FUNCTION_BLOCK FB_AddMcsAxesXyzToMcGroup
VAR_IN_OUT
	stAxis				: ARRAY[1..3] OF AXIS_REF;	
	stGroupRef			: AXES_GROUP_REF;
END_VAR
VAR_INPUT
	bExecute				: BOOL;
END_VAR
VAR_OUTPUT
	bDone				: BOOL;
	bBusy				: BOOL;
	bError				: BOOL;
END_VAR
VAR
	fbAddAxis			: ARRAY[1..3] OF MC_AddAxisToGroup;
	i					: UINT;
END_VAR

bDone := TRUE;
bBusy := FALSE;
bError := FALSE;

fbAddAxis[1].IdentInGroup := MCS_X; //X-Axis
fbAddAxis[2].IdentInGroup := MCS_Y; //Y-Axis
fbAddAxis[3].IdentInGroup := MCS_Z; //Z-Axis

FOR i:=1 TO 3 DO
	fbAddAxis[i](AxesGroup:=stGroupRef, Axis := stAxis[i], Execute := bExecute);

	IF (NOT fbAddAxis[i].Done) THEN
		bDone := FALSE;
	END_IF
	IF (fbAddAxis[i].Busy) THEN
		bBusy := TRUE;
	END_IF
	IF (fbAddAxis[i].Error) THEN
		bError := TRUE;
	END_IF
END_FOR

END_FUNCTION_BLOCK

(* stored: Version 1.1.0.1, ProductVersion 3.1.4024.5
   POU FB_AddMcsAxesXyzToMcGroup: Id {82897557-630f-42f2-9dc0-c94f0234539c}, SpecialFunc None *)
